SYSTEM RMT_DEV_TEST (* RMT_DEV Test with FB_ADD_REAL and E_CTU *)
  (* Standard: 61499 Feasibility Demo ITA *)
  (* Version 0.5, 2001-06-05, JHC, Rockwell Automation, Changed GUI to IN_ANY, OUT_ANY. *)
  (* Version 0.4, 2001-05-22, JHC, Rockwell Automation, Corrected UDP addresses. *)
  (* Version 0.3, 2001-04-26, JHC, Rockwell Automation, Added TEST1, TEST2 applications. *)
  (* Version 0.2, 2001-02-21, JHC, Rockwell Automation, Made all UDP sockets on 224.0.0.1 to work offline. *)
  (* Version 0.1, 2001-01-05, JHC, Rockwell Automation, Added remote counter *)
  (* Version 0.0, 2001-01-03, JHC, Rockwell Automation *)
  APPLICATION TEST1 (* FB_ADD_REAL test *)
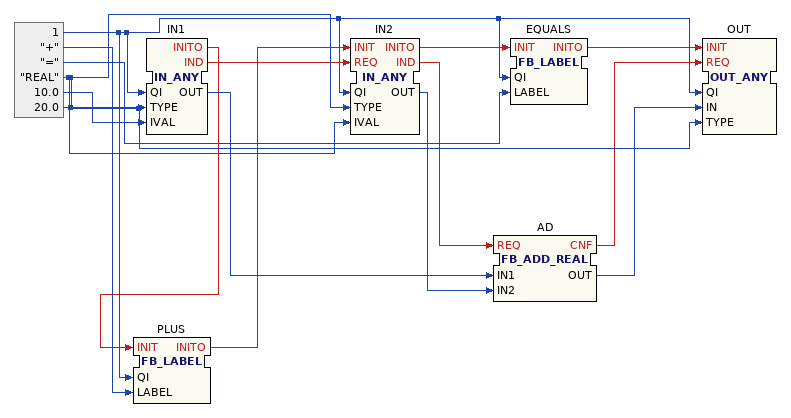
    FBS
      IN1 : IN_ANY;
      PLUS : FB_LABEL;
      IN2 : IN_ANY;
      AD : FB_ADD_REAL;
      EQUALS : FB_LABEL;
      OUT : OUT_ANY;
    END_FBS
    EVENT_CONNECTIONS
      IN1.INITO TO PLUS.INIT;
      PLUS.INITO TO IN2.INIT;
      IN2.INITO TO EQUALS.INIT;
      EQUALS.INITO TO OUT.INIT;
      IN1.IND TO IN2.REQ;
      IN2.IND TO AD.REQ;
      AD.CNF TO OUT.REQ;
    END_CONNECTIONS
    DATA_CONNECTIONS
      1 TO IN1.QI;
      1 TO IN2.QI;
      1 TO OUT.QI;
      1 TO PLUS.QI;
      1 TO EQUALS.QI;
      "+" TO PLUS.LABEL;
      "=" TO EQUALS.LABEL;
      IN1.OUT TO AD.IN1;
      IN2.OUT TO AD.IN2;
      AD.OUT TO OUT.IN;
      "REAL" TO IN1.TYPE;
      "REAL" TO IN2.TYPE;
      "REAL" TO OUT.TYPE;
      10.0 TO IN1.IVAL;
      20.0 TO IN2.IVAL;
    END_CONNECTIONS
  END_APPLICATION
  APPLICATION TEST2 (* E_CTU test *)
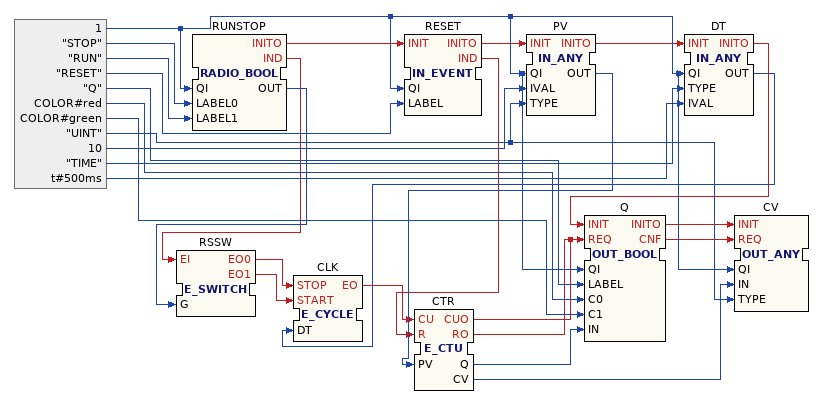
    FBS
      RUNSTOP : RADIO_BOOL;
      RESET : IN_EVENT;
      PV : IN_ANY;
      DT : IN_ANY;
      RSSW : E_SWITCH;
      CLK : E_CYCLE;
      CTR : E_CTU;
      Q : OUT_BOOL;
      CV : OUT_ANY;
    END_FBS
    EVENT_CONNECTIONS
      RUNSTOP.INITO TO RESET.INIT;
      RESET.INITO TO PV.INIT;
      PV.INITO TO DT.INIT;
      DT.INITO TO Q.INIT;
      Q.INITO TO CV.INIT;
      RUNSTOP.IND TO RSSW.EI;
      RSSW.EO0 TO CLK.STOP;
      RSSW.EO1 TO CLK.START;
      CLK.EO TO CTR.CU;
      RESET.IND TO CTR.R;
      CTR.CUO TO Q.REQ;
      CTR.RO TO Q.REQ;
      Q.CNF TO CV.REQ;
    END_CONNECTIONS
    DATA_CONNECTIONS
      1 TO CV.QI;
      1 TO DT.QI;
      1 TO PV.QI;
      1 TO Q.QI;
      1 TO RESET.QI;
      1 TO RUNSTOP.QI;
      "STOP" TO RUNSTOP.LABEL0;
      "RUN" TO RUNSTOP.LABEL1;
      "RESET" TO RESET.LABEL;
      "Q" TO Q.LABEL;
      COLOR#red TO Q.C0;
      COLOR#green TO Q.C1;
      RUNSTOP.OUT TO RSSW.G;
      PV.OUT TO CTR.PV;
      DT.OUT TO CLK.DT;
      CTR.Q TO Q.IN;
      CTR.CV TO CV.IN;
      "UINT" TO CV.TYPE;
      10 TO PV.IVAL;
      "UINT" TO PV.TYPE;
      "TIME" TO DT.TYPE;
      t#500ms TO DT.IVAL;
    END_CONNECTIONS
  END_APPLICATION
  DEVICE DEV_TESTER : FRAME_DEVICE
    RESOURCE RES1 : PANEL_RESOURCE
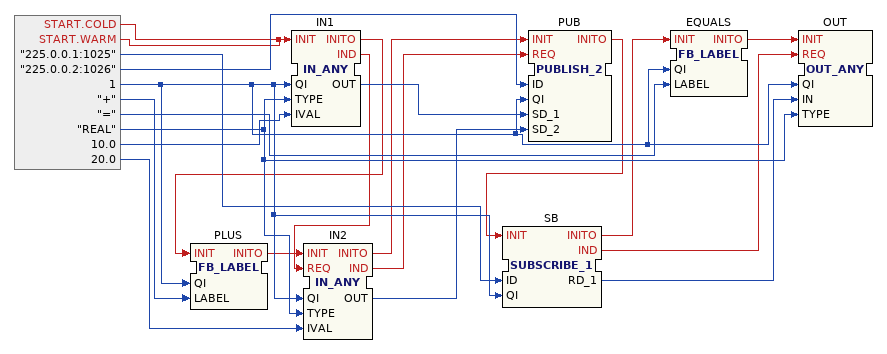
      FBS
        IN1 : IN_ANY;
        PLUS : FB_LABEL;
        IN2 : IN_ANY;
        PUB : PUBLISH_2;
        SB : SUBSCRIBE_1;
        EQUALS : FB_LABEL;
        OUT : OUT_ANY;
      END_FBS
      EVENT_CONNECTIONS
        START.COLD TO IN1.INIT;
        START.WARM TO IN1.INIT;
        IN1.INITO TO PLUS.INIT;
        PLUS.INITO TO IN2.INIT;
        IN2.INITO TO PUB.INIT;
        PUB.INITO TO SB.INIT;
        SB.INITO TO EQUALS.INIT;
        EQUALS.INITO TO OUT.INIT;
        IN1.IND TO IN2.REQ;
        IN2.IND TO PUB.REQ;
        SB.IND TO OUT.REQ;
      END_CONNECTIONS
      DATA_CONNECTIONS
        "225.0.0.1:1025" TO SB.ID;
        "225.0.0.2:1026" TO PUB.ID;
        1 TO IN1.QI;
        1 TO IN2.QI;
        1 TO PUB.QI;
        1 TO SB.QI;
        1 TO OUT.QI;
        1 TO PLUS.QI;
        1 TO EQUALS.QI;
        "+" TO PLUS.LABEL;
        "=" TO EQUALS.LABEL;
        IN1.OUT TO PUB.SD_1;
        IN2.OUT TO PUB.SD_2;
        SB.RD_1 TO OUT.IN;
        "REAL" TO IN1.TYPE;
        "REAL" TO IN2.TYPE;
        "REAL" TO OUT.TYPE;
        10.0 TO IN1.IVAL;
        20.0 TO IN2.IVAL;
      END_CONNECTIONS
    END_RESOURCE
    RESOURCE RES2 : PANEL_RESOURCE
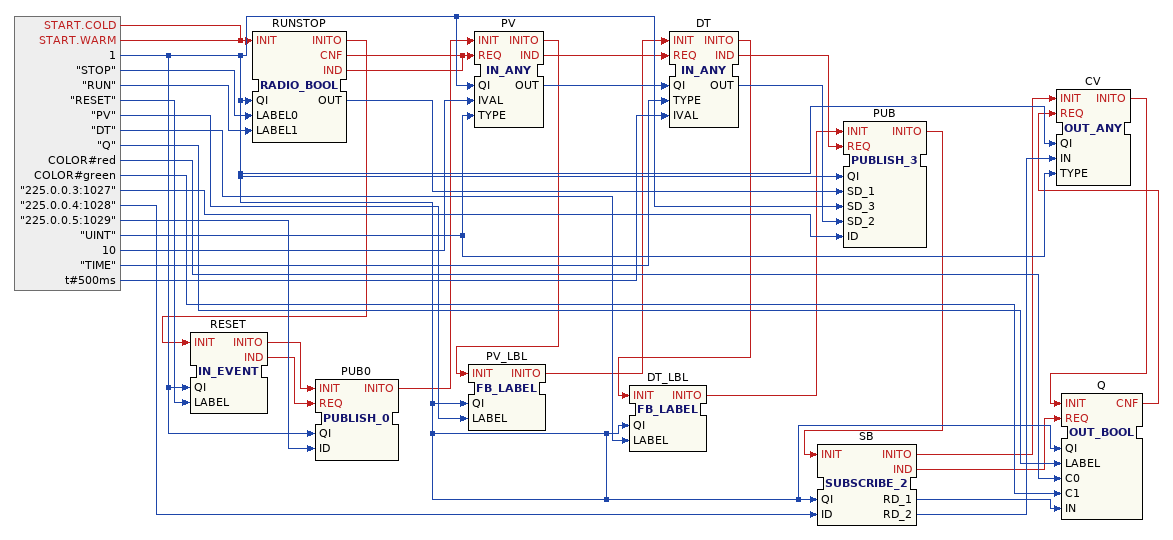
      FBS
        RUNSTOP : RADIO_BOOL;
        RESET : IN_EVENT;
        PUB0 : PUBLISH_0;
        PV : IN_ANY;
        PV_LBL : FB_LABEL;
        DT : IN_ANY;
        DT_LBL : FB_LABEL;
        PUB : PUBLISH_3;
        SB : SUBSCRIBE_2;
        Q : OUT_BOOL;
        CV : OUT_ANY;
      END_FBS
      EVENT_CONNECTIONS
        START.COLD TO RUNSTOP.INIT;
        START.WARM TO RUNSTOP.INIT;
        RUNSTOP.INITO TO RESET.INIT;
        RESET.INITO TO PUB0.INIT;
        PUB0.INITO TO PV.INIT;
        PV.INITO TO PV_LBL.INIT;
        PV_LBL.INITO TO DT.INIT;
        DT.INITO TO DT_LBL.INIT;
        DT_LBL.INITO TO PUB.INIT;
        PUB.INITO TO SB.INIT;
        SB.INITO TO CV.INIT;
        CV.INITO TO Q.INIT;
        RUNSTOP.CNF TO PV.REQ;
        RUNSTOP.IND TO PV.REQ;
        RESET.IND TO PUB0.REQ;
        PV.IND TO DT.REQ;
        DT.IND TO PUB.REQ;
        SB.IND TO Q.REQ;
        Q.CNF TO CV.REQ;
      END_CONNECTIONS
      DATA_CONNECTIONS
        1 TO CV.QI;
        1 TO DT.QI;
        1 TO PUB.QI;
        1 TO PUB0.QI;
        1 TO PV.QI;
        1 TO Q.QI;
        1 TO RESET.QI;
        1 TO RUNSTOP.QI;
        1 TO SB.QI;
        1 TO PV_LBL.QI;
        1 TO DT_LBL.QI;
        "STOP" TO RUNSTOP.LABEL0;
        "RUN" TO RUNSTOP.LABEL1;
        "RESET" TO RESET.LABEL;
        "PV" TO PV_LBL.LABEL;
        "DT" TO DT_LBL.LABEL;
        "Q" TO Q.LABEL;
        COLOR#red TO Q.C0;
        COLOR#green TO Q.C1;
        RUNSTOP.OUT TO PUB.SD_1;
        PV.OUT TO PUB.SD_3;
        DT.OUT TO PUB.SD_2;
        SB.RD_1 TO Q.IN;
        SB.RD_2 TO CV.IN;
        "225.0.0.3:1027" TO PUB.ID;
        "225.0.0.4:1028" TO SB.ID;
        "225.0.0.5:1029" TO PUB0.ID;
        "UINT" TO CV.TYPE;
        10 TO PV.IVAL;
        "UINT" TO PV.TYPE;
        "TIME" TO DT.TYPE;
        t#500ms TO DT.IVAL;
      END_CONNECTIONS
    END_RESOURCE
    DATA_CONNECTIONS
      1 TO RES1.TRACE;
    END_CONNECTIONS
  END_DEVICE
  DEVICE DEV1 : RMT_DEV
    RESOURCE RES1 : EMB_RES
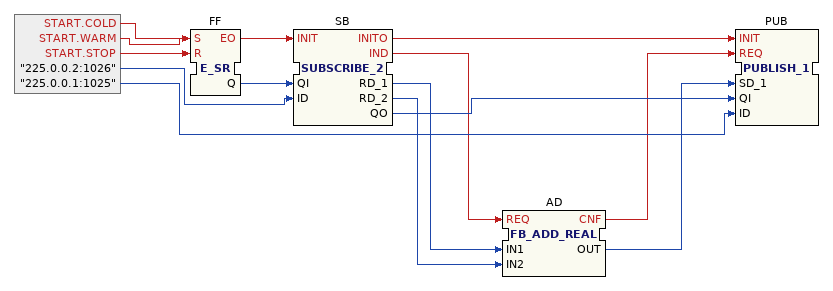
      FBS
        FF : E_SR;
        SB : SUBSCRIBE_2;
        AD : FB_ADD_REAL;
        PUB : PUBLISH_1;
      END_FBS
      EVENT_CONNECTIONS
        START.COLD TO FF.S;
        START.WARM TO FF.S;
        START.STOP TO FF.R;
        FF.EO TO SB.INIT;
        SB.INITO TO PUB.INIT;
        SB.IND TO AD.REQ;
        AD.CNF TO PUB.REQ;
      END_CONNECTIONS
      DATA_CONNECTIONS
        SB.RD_1 TO AD.IN1;
        SB.RD_2 TO AD.IN2;
        AD.OUT TO PUB.SD_1;
        FF.Q TO SB.QI;
        SB.QO TO PUB.QI;
        "225.0.0.2:1026" TO SB.ID;
        "225.0.0.1:1025" TO PUB.ID;
      END_CONNECTIONS
    END_RESOURCE
    RESOURCE RES2 : EMB_RES
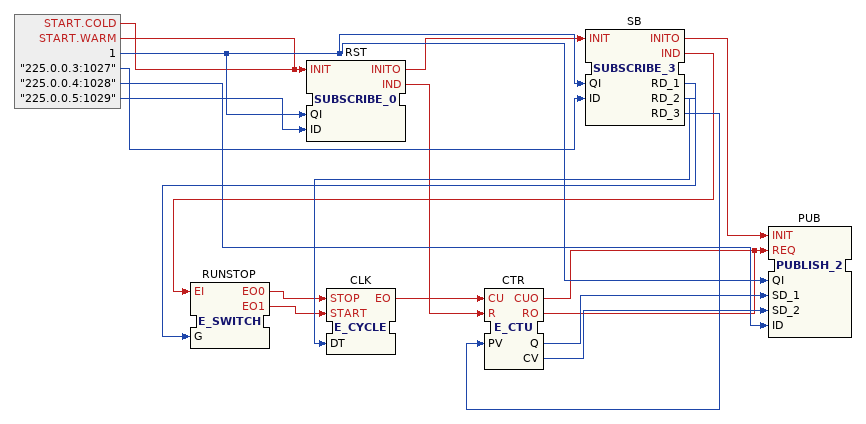
      FBS
        SB : SUBSCRIBE_3;
        RST : SUBSCRIBE_0;
        RUNSTOP : E_SWITCH;
        CLK : E_CYCLE;
        CTR : E_CTU;
        PUB : PUBLISH_2;
      END_FBS
      EVENT_CONNECTIONS
        START.COLD TO RST.INIT;
        START.WARM TO RST.INIT;
        RST.INITO TO SB.INIT;
        SB.INITO TO PUB.INIT;
        SB.IND TO RUNSTOP.EI;
        RUNSTOP.EO0 TO CLK.STOP;
        RUNSTOP.EO1 TO CLK.START;
        CLK.EO TO CTR.CU;
        RST.IND TO CTR.R;
        CTR.CUO TO PUB.REQ;
        CTR.RO TO PUB.REQ;
      END_CONNECTIONS
      DATA_CONNECTIONS
        1 TO PUB.QI;
        1 TO SB.QI;
        1 TO RST.QI;
        SB.RD_1 TO RUNSTOP.G;
        SB.RD_2 TO CLK.DT;
        SB.RD_3 TO CTR.PV;
        CTR.Q TO PUB.SD_1;
        CTR.CV TO PUB.SD_2;
        "225.0.0.3:1027" TO SB.ID;
        "225.0.0.4:1028" TO PUB.ID;
        "225.0.0.5:1029" TO RST.ID;
      END_CONNECTIONS
    END_RESOURCE
  END_DEVICE
  DATA_CONNECTIONS (* parameter values *)
    [50,50,190,250] TO DEV_TESTER.BOUNDS;
    [2,1] TO DEV_TESTER.GRID;
    "localhost:61501" TO DEV1.MGR_ID;
  END_CONNECTIONS
  MAPPINGS
    TEST1.IN1 ON DEV_TESTER.RES1.IN1;
    TEST1.PLUS ON DEV_TESTER.RES1.PLUS;
    TEST1.IN2 ON DEV_TESTER.RES1.IN2;
    TEST1.EQUALS ON DEV_TESTER.RES1.EQUALS;
    TEST1.AD ON DEV1.RES1.AD;
    TEST1.OUT ON DEV_TESTER.RES1.OUT;
    TEST2.RUNSTOP ON DEV_TESTER.RES2.RUNSTOP;
    TEST2.RESET ON DEV_TESTER.RES2.RESET;
    TEST2.PV ON DEV_TESTER.RES2.PV;
    TEST2.DT ON DEV_TESTER.RES2.DT;
    TEST2.RSSW ON DEV1.RES2.RUNSTOP;
    TEST2.CLK ON DEV1.RES2.CLK;
    TEST2.CTR ON DEV1.RES2.CTR;
    TEST2.Q ON DEV_TESTER.RES2.Q;
    TEST2.CV ON DEV_TESTER.RES2.CV;
  END_MAPPINGS
END_SYSTEM
